(* PLC project Unnamed, Unknown Unnamed 1 *)
(* stored: creationDateTime 2026-08-05T10:33:57, modificationDateTime 2026-08-16T13:41:07 *)

PROGRAM program0
  VAR
    systec_out AT %QB0.0.2.25088.1 : USINT := 2#10101010;  (* canfestival_0/CanOpenNode_0/systec_IO-X1/0x6200-0x01: Write Outputs 0x1 to 0x8 *)
    systec_in AT %IB0.0.2.24576.1 : USINT;  (* canfestival_0/CanOpenNode_0/systec_IO-X1/0x6000-0x01: Read Inputs 0x1 to 0x8 *)
    position AT %ID0.0.7.24676.0 : DINT;  (* canfestival_0/CanOpenNode_0/CanOpenCIA402Node_0/0x6064-0x00: Position actual value *)
  END_VAR
  VAR
    position0 : DINT;  (* canfestival_0/CanOpenNode_0/CanOpenCIA402Node_0/0x6064-0x00: Position actual value *)
  END_VAR

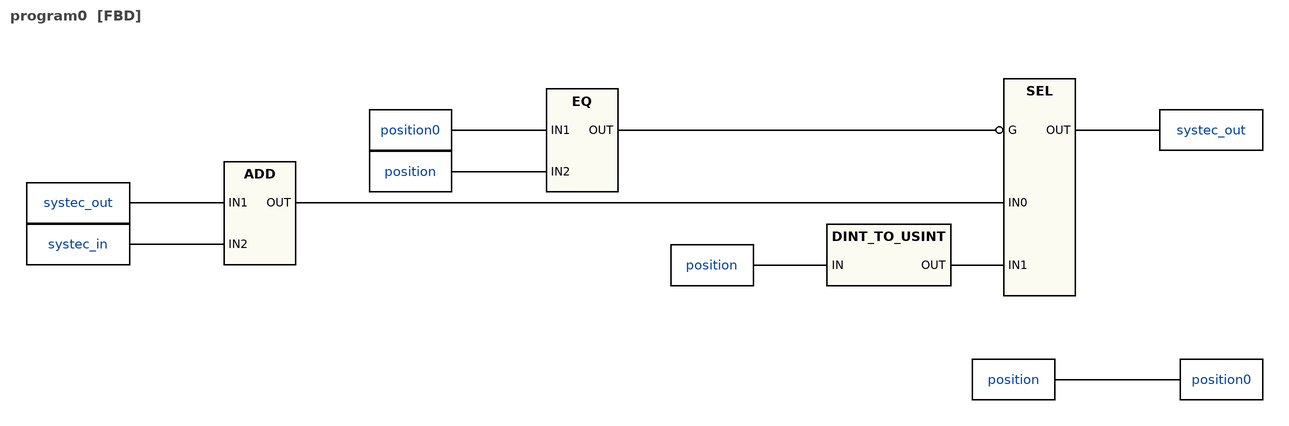
(* FBD diagram, written out as Structured Text *)
systec_out := SEL(NOT (position0 = position), systec_out + systec_in, DINT_TO_USINT(position));
position0 := position;
END_PROGRAM

CONFIGURATION config
  RESOURCE resource1 ON PLC
    TASK task0(INTERVAL := T#20ms, PRIORITY := 0);
    PROGRAM instance0 WITH task0 : program0;
  END_RESOURCE
END_CONFIGURATION
